// TIA Portal project "proj_2" (V21)

(* hardware
DEVICE "S7-1500/ET200MP station_1"  S7-1500 station
   slot 0: "Rail_0"  Rack  6ES7 590-1***0-0AA0
   slot 1: "PLC_1"  CPU 1512C-1 PN  6ES7 512-1CM03-0AB0  V4.1
      slot 3: "CPU display_1"  6ES7591-1AA00-0AA0
      slot 32768: "PROFINET interface_1"  X1
         slot 32769: "Port_1"  X1 P1
         slot 32770: "Port_2"  X1 P2
      slot 34817: "Virtual CP interface port_1"  Virtual CP interface port  Virtual CP interface port FW V4.1
*)

// ===== PLC "PLC_1"  CPU 1512C-1 PN =====

VAR_GLOBAL   // PLC tag table "Inputs"
   "proximity_sw" AT %I0.0 : Bool;
   "level_sw" AT %I0.1 : Bool;
   "red_eye" AT %I0.2 : Bool;
   "blue_eye" AT %I0.3 : Bool;
END_VAR

VAR_GLOBAL   // PLC tag table "Outputs"
   "conveyor_motor" AT %Q0.0 : Bool;
   "walnut_hopper" AT %Q0.1 : Bool;
   "pecan_hopper" AT %Q0.2 : Bool;
END_VAR

// folder: Classes

DATA_BLOCK "conveyor"   // DB1
{ S7_Optimized_Access := 'TRUE' }
VERSION : 0.1
// stored: InstanceOfName START_STOP
"START_STOP"
BEGIN
END_DATA_BLOCK

DATA_BLOCK "sorting_DB"   // DB2
{ S7_Optimized_Access := 'TRUE' }
VERSION : 0.1
// stored: InstanceOfName sorting
"sorting"
BEGIN
END_DATA_BLOCK

// folder: (top level)

FUNCTION_BLOCK "START_STOP"   // FB1, SCL
{ S7_Optimized_Access := 'TRUE' }
VERSION : 0.1
   VAR_INPUT
      start : Bool;
      stop : Bool;
   END_VAR
   VAR_OUTPUT
      device_on : Bool;
   END_VAR
   VAR
      start_ons : R_TRIG;
      stop_ons : R_TRIG;
   END_VAR
BEGIN
   //this is like a class
   #start_ons(CLK:=#start);
   #stop_ons(CLK := #stop);




   IF #start_ons.Q THEN
       #device_on := TRUE;
   END_IF;

   IF #stop_ons.Q THEN
       #device_on := false;
   END_IF;
END_FUNCTION_BLOCK

FUNCTION_BLOCK "sorting"   // FB2, SCL
{ S7_Optimized_Access := 'TRUE' }
VERSION : 0.1
   VAR_INPUT
      sort_start : Bool;
      sort_1 : Bool;
      sort_2 : Bool;
   END_VAR
   VAR_OUTPUT
      actuator_1 : Bool;
      actuator_2 : Bool;
   END_VAR
   VAR
      filter : TON_TIME;
   END_VAR
BEGIN
   #filter(IN := #sort_start,
                         PT := T#200ms);


   IF #filter.Q THEN
       IF #sort_1 THEN
           #actuator_1 := true;
       ELSIF #sort_2 THEN
           #actuator_2 := true;
       ELSE
           #actuator_1 := FALSE;
           #actuator_2 := FALSE;
       END_IF;
   END_IF;
END_FUNCTION_BLOCK

ORGANIZATION_BLOCK "Main"   // OB1, LAD, ProgramCycle
TITLE = "Main Program Sweep (Cycle)"
{ S7_Optimized_Access := 'TRUE' }
VERSION : 0.1
   VAR_INPUT
      Initial_Call : Bool;   // Initial call of this OB
      Remanence : Bool;   // =True, if remanent data are available
   END_VAR
BEGIN
END_ORGANIZATION_BLOCK

ORGANIZATION_BLOCK "Main_scl"   // OB123, SCL, ProgramCycle
TITLE = "Main Program Sweep (Cycle)"
{ S7_Optimized_Access := 'TRUE' }
VERSION : 0.1
   VAR_INPUT
      Initial_Call : Bool;   // Initial call of this OB
      Remanence : Bool;   // =True, if remanent data are available
   END_VAR
   VAR_TEMP
      conveyor_motor_bit : Bool;
      pecan_hopper_bit : Bool;
      walnut_hopper_bit : Bool;
   END_VAR
BEGIN
   "conveyor"(start:=NOT "proximity_sw" OR ("proximity_sw" AND "level_sw"),
              stop:="proximity_sw",
              device_on=>#conveyor_motor_bit);


   "sorting_DB"(sort_start:="proximity_sw",
                sort_1:="on_until"("red_eye" AND NOT "level_sw"),
                sort_2:="on_until"("blue_eye" AND NOT "level_sw"),
                actuator_1=>#pecan_hopper_bit,
                actuator_2=>#walnut_hopper_bit);

   //outputs
   "conveyor_motor" := #conveyor_motor_bit;
   "pecan_hopper" := #pecan_hopper_bit;
   "walnut_hopper" := #walnut_hopper_bit;
END_ORGANIZATION_BLOCK

// folder: functions

FUNCTION "sensor_true" : Bool   // FC1, SCL
{ S7_Optimized_Access := 'TRUE' }
VERSION : 0.1
   VAR_INPUT
      sensor : Bool;
   END_VAR
BEGIN
   IF #sensor THEN
       #sensor_true := TRUE;
   ELSE
       #sensor_true := false;
   END_IF;
END_FUNCTION

FUNCTION "on_until" : Bool   // FC2, SCL
{ S7_Optimized_Access := 'TRUE' }
VERSION : 0.1
   VAR_INPUT
      on_condition : Bool;
   END_VAR
BEGIN
   IF #on_condition THEN
       #on_until := TRUE;
   ELSE
       #on_until := FALSE;
   END_IF;
END_FUNCTION